// TIA Portal V18 export
ORGANIZATION_BLOCK "Main"   // OB1, LAD, ProgramCycle
TITLE = "Main Program Sweep (Cycle)"
{ S7_Optimized_Access := 'TRUE' }
VERSION : 0.1
// stored: AutoNumber true, IsIECCheckEnabled false, SetENOAutomatically false
   VAR_INPUT
      Initial_Call : Bool;   // Initial call of this OB
      Remanence : Bool;   // =True, if remanent data are available
   END_VAR
BEGIN

REGION Network 1
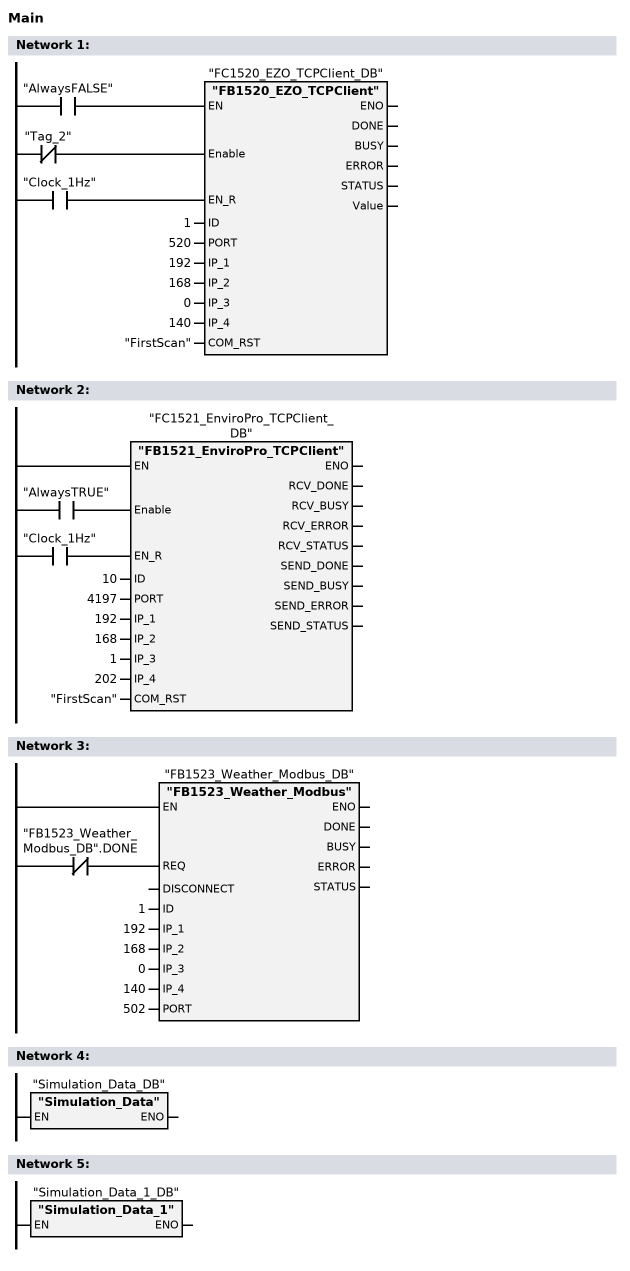
   RUNG wire#powerrail
      Contact( "AlwaysFALSE" )
      "FC1520_EZO_TCPClient_DB"(Enable := wire#w1, EN_R := wire#w2, ID := 1, PORT := 520, IP_1 := 192, IP_2 := 168, IP_3 := 0, IP_4 := 140, COM_RST := "FirstScan", DONE =>, BUSY =>, ERROR =>, STATUS =>, Value =>)
   END_RUNG
   RUNG wire#powerrail
      I_Contact( "Tag_2" )
   END_RUNG wire#w1
   RUNG wire#powerrail
      Contact( "Clock_1Hz" )
   END_RUNG wire#w2
   // the same network as SCL:
   IF "AlwaysFALSE" THEN
       "FC1520_EZO_TCPClient_DB"(Enable := NOT "Tag_2",   // "FB1520_EZO_TCPClient"
                               EN_R := "Clock_1Hz",
                               ID := 1,
                               PORT := 520,
                               IP_1 := 192,
                               IP_2 := 168,
                               IP_3 := 0,
                               IP_4 := 140,
                               COM_RST := "FirstScan");
   END_IF;
END_REGION

REGION Network 2
   RUNG wire#powerrail
      "FC1521_EnviroPro_TCPClient_DB"(Enable := wire#w1, EN_R := wire#w2, ID := 10, PORT := 4197, IP_1 := 192, IP_2 := 168, IP_3 := 1, IP_4 := 202, COM_RST := "FirstScan", RCV_DONE =>, RCV_BUSY =>, RCV_ERROR =>, RCV_STATUS =>, SEND_DONE =>, SEND_BUSY =>, SEND_ERROR =>, SEND_STATUS =>)
   END_RUNG
   RUNG wire#powerrail
      Contact( "AlwaysTRUE" )
   END_RUNG wire#w1
   RUNG wire#powerrail
      Contact( "Clock_1Hz" )
   END_RUNG wire#w2
   // the same network as SCL:
   "FC1521_EnviroPro_TCPClient_DB"(Enable := "AlwaysTRUE",   // "FB1521_EnviroPro_TCPClient"
                           EN_R := "Clock_1Hz",
                           ID := 10,
                           PORT := 4197,
                           IP_1 := 192,
                           IP_2 := 168,
                           IP_3 := 1,
                           IP_4 := 202,
                           COM_RST := "FirstScan");
END_REGION

REGION Network 3
   RUNG wire#powerrail
      "FB1523_Weather_Modbus_DB"(REQ := wire#w1, DISCONNECT :=, ID := 1, IP_1 := 192, IP_2 := 168, IP_3 := 0, IP_4 := 140, PORT := 502, DONE =>, BUSY =>, ERROR =>, STATUS =>)
   END_RUNG
   RUNG wire#powerrail
      I_Contact( "FB1523_Weather_Modbus_DB".DONE )
   END_RUNG wire#w1
   // the same network as SCL:
   "FB1523_Weather_Modbus_DB"(REQ := NOT "FB1523_Weather_Modbus_DB".DONE,   // "FB1523_Weather_Modbus"
                           ID := 1,
                           IP_1 := 192,
                           IP_2 := 168,
                           IP_3 := 0,
                           IP_4 := 140,
                           PORT := 502);
END_REGION

REGION Network 4
   RUNG wire#powerrail
      "Simulation_Data_DB"()
   END_RUNG
   // the same network as SCL:
   "Simulation_Data_DB"();   // "Simulation_Data"
END_REGION

REGION Network 5
   RUNG wire#powerrail
      "Simulation_Data_1_DB"()
   END_RUNG
   // the same network as SCL:
   "Simulation_Data_1_DB"();   // "Simulation_Data_1"
END_REGION
END_ORGANIZATION_BLOCK
